# EPICS substitutions: ni9239ethdaqApp/Db/ni9239acq.substitutions
file db/ni9239acqperchannel.db {
    pattern{CH, BPMCH}
    {"0", "A"}
    {"1", "C"}
    {"2", "B"}
    {"3", "D"}
}
